ABB RobotStudio station: Simulation_miniproject.rsstn

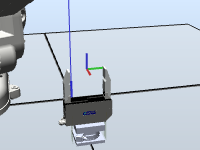
Station Simulation_miniproject (saved by RobotStudio 6.6.7701.1025)
Controller Matlab_tcp, task T_ROB1: task frame (RAPID world) sits at (0, -395.13, 0) mm in the station
Controller Matlab_tcp
  mechanical unit ROB_1: IRB140_6_81_C_03, 6 joints, base frame (0, 0, 0) mm
Layout (positions relative to the parent item):
  - IRB140_6_81_C_03 [mechanism, from Robots\IRB140_6_81_C_G_03.rslib] at (0, -395.13, 0) mm; joint values [0.4324, 1.0224, -1.4931, -0.4248, 1.0769, 0.438] (rad or m)
  - SmartComponent_1 [smart component, from Libraries\Workshop_gripper.rslib]
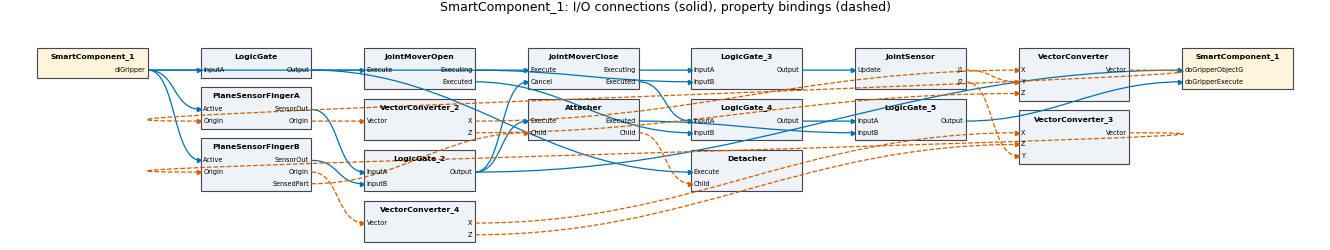
      connections:
        SmartComponent_1.diGripper -> LogicGate.InputA
        SmartComponent_1.diGripper -> PlaneSensorFingerA.Active
        SmartComponent_1.diGripper -> PlaneSensorFingerB.Active
        PlaneSensorFingerA.SensorOut -> LogicGate_2.InputA
        PlaneSensorFingerB.SensorOut -> LogicGate_2.InputB
        SmartComponent_1.diGripper -> JointMoverClose.Execute
        LogicGate_2.Output -> JointMoverClose.Cancel
        LogicGate_2.Output -> SmartComponent_1.doGripperObjectGrasped
        LogicGate.Output -> JointMoverOpen.Execute
        JointMoverClose.Executing -> LogicGate_3.InputA
        JointMoverOpen.Executing -> LogicGate_3.InputB
        LogicGate_3.Output -> JointSensor.Update
        LogicGate_2.Output -> Attacher.Execute
        LogicGate.Output -> Detacher.Execute
        JointMoverClose.Executed -> LogicGate_4.InputA
        JointMoverOpen.Executed -> LogicGate_4.InputB
        LogicGate_4.Output -> LogicGate_5.InputA
        Attacher.Executed -> LogicGate_5.InputB
        LogicGate_5.Output -> SmartComponent_1.doGripperExecuted
        VectorConverter_2.X => VectorConverter.X
        JointSensor.J1 => VectorConverter.Y
        VectorConverter_2.Z => VectorConverter.Z
        VectorConverter.Vector => PlaneSensorFingerA.Origin
        PlaneSensorFingerA.Origin => VectorConverter_2.Vector
        VectorConverter_4.X => VectorConverter_3.X
        VectorConverter_4.Z => VectorConverter_3.Z
        JointSensor.J2 => VectorConverter_3.Y
        VectorConverter_3.Vector => PlaneSensorFingerB.Origin
        PlaneSensorFingerB.Origin => VectorConverter_4.Vector
        PlaneSensorFingerB.SensedPart => Attacher.Child
        Attacher.Child => Detacher.Child
    - SCHUNK_WSG_GRIPPER [mechanism, from Libraries\Workshop_gripper.rslib] at (0, 0, 0) mm; joint values [0.0535, -0.0535] (rad or m)
    - PlaneSensorFingerA [smart component, from Components\PlaneSensor.rslib] at (300, 0, 0) mm
        properties: Origin=[0 0.0535 0]; Axis1=[0.03 0 0]; Axis2=[0 0 0.099]; SensedPart=(none)
      - _sensorPart_ [part, from Libraries\Workshop_gripper.rslib]
    - PlaneSensorFingerB [smart component, from Components\PlaneSensor.rslib] at (300, 0, 0) mm
        properties: Origin=[0 -0.0535 0]; Axis1=[0.03 0 0]; Axis2=[0 0 0.099]; SensedPart=(none)
      - _sensorPart_ [part, from Libraries\Workshop_gripper.rslib]
    - JointMoverClose [smart component, from Components\JointMover.rslib]
        properties: Mechanism=SCHUNK_WSG_GRIPPER; Relative=false; Duration=2; J1=0.0535; J2=-0.0535
    - JointMoverOpen [smart component, from Components\JointMover.rslib]
        properties: Mechanism=SCHUNK_WSG_GRIPPER; Relative=false; Duration=2; J1=0.0535; J2=-0.0535
    - LogicGate [smart component, from Components\LogicGate.rslib]
        properties: Operator=NOT; Delay=0
    - LogicGate_2 [smart component, from Components\LogicGate.rslib]
        properties: Operator=AND; Delay=0
    - JointSensor [smart component, from Components\JointSensor.rslib]
        properties: Mechanism=SCHUNK_WSG_GRIPPER; J1=0.0535; J2=-0.0535
    - LogicGate_3 [smart component, from Components\LogicGate.rslib]
        properties: Operator=OR; Delay=0
    - VectorConverter [smart component, from Components\VectorConverter.rslib]
        properties: X=0; Y=0.0535; Z=0; Vector=[0 0.0535 0]
    - VectorConverter_2 [smart component, from Components\VectorConverter.rslib]
        properties: X=0; Y=0.0535; Z=0; Vector=[0 0.0535 0]
    - VectorConverter_3 [smart component, from Components\VectorConverter.rslib]
        properties: X=0; Y=-0.0535; Z=0; Vector=[0 -0.0535 0]
    - VectorConverter_4 [smart component, from Components\VectorConverter.rslib]
        properties: X=0; Y=-0.0535; Z=0; Vector=[0 -0.0535 0]
    - Attacher [smart component, from Components\Attacher.rslib]
        properties: Parent=SCHUNK_WSG_GRIPPER; Flange=0; Child=(none); Mount=false; Offset=[0 0 0]; Orientation=[0 0 0]
    - Detacher [smart component, from Components\Detacher.rslib]
        properties: Child=(none); KeepPosition=true
    - LogicGate_4 [smart component, from Components\LogicGate.rslib]
        properties: Operator=OR; Delay=0
    - LogicGate_5 [smart component, from Components\LogicGate.rslib]
        properties: Operator=OR; Delay=0
  - SCHUNK_body_gripper [part] at (300, 0, 0) mm
    - SCHUNK_WSG_GRIPPER_1 [frame] at (0, 0, 234.82) mm
  - SCHUNK_fingerA [part] at (300, 0, 0) mm
  - SCHUNK_fingerB [part] at (300, 0, 0) mm
Targets, tools, work objects and paths stored in the station, written as RAPID:
! task T_ROB1
MODULE FunctionHandler
  PERS tooldata defaultTool:=[TRUE,[[0,0,0],[1,0,0,0]],[1,[0,0,0.001],[1,0,0,0],0,0,0]];
  PERS wobjdata defaultWobj:=[FALSE,TRUE,"",[[0,395.127094574,0],[1,0,0,0]],[[0,0,0],[1,0,0,0]]];
  VAR signaldo defaultTakePictureActivationIO;
  VAR signaldi defaultTakePictureExecutedIO;
  PROC FH_TakePicture()
    SetDO defaultTakePictureActivationIO,1;
    WaitDI defaultTakePictureExecutedIO,1;
    SetDO defaultTakePictureActivationIO,0;
  ENDPROC
ENDMODULE

! task T_ROB1
MODULE CommandHandler
  PROC COMH_CommandListener()
  ENDPROC
ENDMODULE

! task T_ROB1
MODULE Thorsten_simulering
  PROC main()
    IP_Initialize;
    COMH_CommandListener;
  ENDPROC
ENDMODULE

! task T_ROB1
MODULE InitParameters
  PROC IP_Initialize()
    ConfL \Off;
    ConfJ \Off;
  ENDPROC
ENDMODULE

! task T_ROB1
MODULE CalibData
  PERS tooldata Servo:=[TRUE,[[0,0,84],[1,0,0,0]],[0.226,[8.9,12.3,48.7],[1,0,0,0],0.00021,0.00024,0.00009]];
  PERS tooldata VaccumOne:=[TRUE,[[56,18.5,37.5],[0.707106781,0,0.707106781,0]],[0.226,[8.9,12.3,48.7],[1,0,0,0],0.00021,0.00024,0.00009]];
ENDMODULE

